// Mitsubishi GX Works2 project: PLCֹ_GROUP_20   PLC: FX3G

// global labels: Global1
VAR_GLOBAL
  Start_Day AT X010 : BOOL;
  Work_Day_Lamp AT Y010 : BOOL;
  Flour_Input AT D1100 : REAL;
  Yeast_Input AT D1110 : REAL;
  Water_Input AT D1120 : REAL;
  Oil_input AT D1130 : REAL;
  Spice_Input AT D1140 : REAL;
  Flour_Container AT D1150 : REAL;
  Yeast_Container AT D1160 : REAL;
  Water_Container AT D1170 : REAL;
  Oil_Container AT D1180 : REAL;
  Spice_Container AT D1190 : REAL;
  Flour_Constant AT E100 : REAL;
  Empty_Flour AT M1 : BOOL;
  Yeast_Ratio AT E0.2 : REAL;
  Water_Ratio AT E0.5 : REAL;
  Oil_Ratio AT E0.3 : REAL;
  Spice_Ratio AT E0.1 : REAL;
  Yeast_Flour_Ratio AT D1200 : REAL;
  Water_Flour_Ratio AT D1210 : REAL;
  Oil_Flour_Ratio AT D1220 : REAL;
  Spice_Flour_Ratio AT D1230 : REAL;
  Out_Of_Stock AT M3 : BOOL;
  Emergency_Stop AT X007 : BOOL;
  End_Of_Day AT M5 : BOOL;
  Const_3secs AT K30 : WORD;
  TC_1 AT TC1 : BOOL;
  TC_3 AT TC3 : BOOL;
  TC_5 AT TC5 : BOOL;
  TS_1 AT TS1 : BOOL;
  TS_5 AT TS5 : BOOL;
  TS_3 AT TS3 : BOOL;
  const_hazi AT K5 : INT;
  TS_9 AT TS9 : BOOL;
  TS_10 AT TS10 : BOOL;
  TS_11 AT TS11 : BOOL;
  TC_9 AT TC9 : BOOL;
  TC_11 AT TC11 : BOOL;
  TC_10 AT TC10 : BOOL;
  Flicker_3secs AT M100 : BOOL;
  Start_Loading_Process AT X002 : BOOL;
  Timer_3s AT TC3 : BOOL;
  Timer_3s_const AT K30 : INT;
  Preparing_Light AT Y005 : BOOL;
  Const_30_Oil AT E30.0 : REAL;
  Const_10_Spice AT E10.0 : REAL;
  Const_100_Flour AT E100.0 : REAL;
  Const_20_Yeast AT E20.0 : REAL;
  Const_50_Water AT E50.0 : REAL;
  Oil_Scale AT D3500 : REAL;
  Spice_Scale AT D3600 : REAL;
  Flour_Scale AT D3200 : REAL;
  Yeast_Scale AT D3300 : REAL;
  Water_Scale AT D3400 : REAL;
  Timer_3s_TS3 AT TS3 : BOOL;
  Kneading_Lamp AT Y001 : BOOL;
  Start_Kneading AT X001 : BOOL;
  Const_210 AT E210.0 : REAL;
  D_Kneading AT D3700 : REAL;
  Start_Proofing AT X011 : BOOL;
  Click_Counter AT CC1 : BOOL;
  Clicks AT K2 : INT;
  Clicks2 AT CS1 : BOOL;
  TC_4 AT TC4 : BOOL;
  Timer_3sec AT K30 : INT;
  Finish_Timer AT TS4 : BOOL;
  Start_Blink AT M300 : BOOL;
  Timer_Blink3 AT K3 : INT;
  Y2_timer AT TS5 : BOOL;
  Lamp_2 AT Y002 : BOOL;
  Lamp_3 AT Y003 : BOOL;
  TC_6 AT TC6 : BOOL;
  Y3_timer AT TS6 : BOOL;
  Finish_Proofing AT M301 : BOOL;
  D_Proofing AT D6000 : REAL;
  Baking_Timer AT TC20 : BOOL;
  Timer_4Secs AT K40 : INT;
  Baking_Lamp AT Y004 : BOOL;
  Y4_Timer AT TS20 : BOOL;
  D_Oven AT D7000 : REAL;
  Checking_Quality AT X003 : BOOL;
  Analog_Input_2 AT D8281 : INT;
  Save_Analog AT D1700 : REAL;
  Const_400 AT E400.0 : REAL;
  Norm_Input AT D1900 : REAL;
  Const_5 AT E2000.0 : REAL;
  Const_1 AT E400.0 : REAL;
  LT_5 AT M123 : BOOL;
  GT_1 AT M127 : BOOL;
  Quality_Lamp AT Y006 : BOOL;
  Timer_5secs AT TC18 : BOOL;
  Timer_5sec AT TS18 : BOOL;
  Const_555 AT K50 : INT;
  D_Shelf AT D5555 : REAL;
  Process_Done AT M63 : BOOL;
  Check_Counter AT CC5 : BOOL;
  Check_Clickes AT K2 : INT;
  Checks AT K2 : INT;
  False_Quality AT M96 : BOOL;
  Quality_Clicks AT CS5 : BOOL;
  Turn_Off_Y1 AT M275 : BOOL;
  Keep_Y1_Work_Right AT M201 : BOOL;
END_VAR

// task Task_01 (event TRUE, interval 0, priority 31): POU_01

PROGRAM POU_01
(* structured ladder/FBD written out as ST: instructions are called as NAME(EN, inputs, outputs); _pN, _eN, _tN stand for wires *)
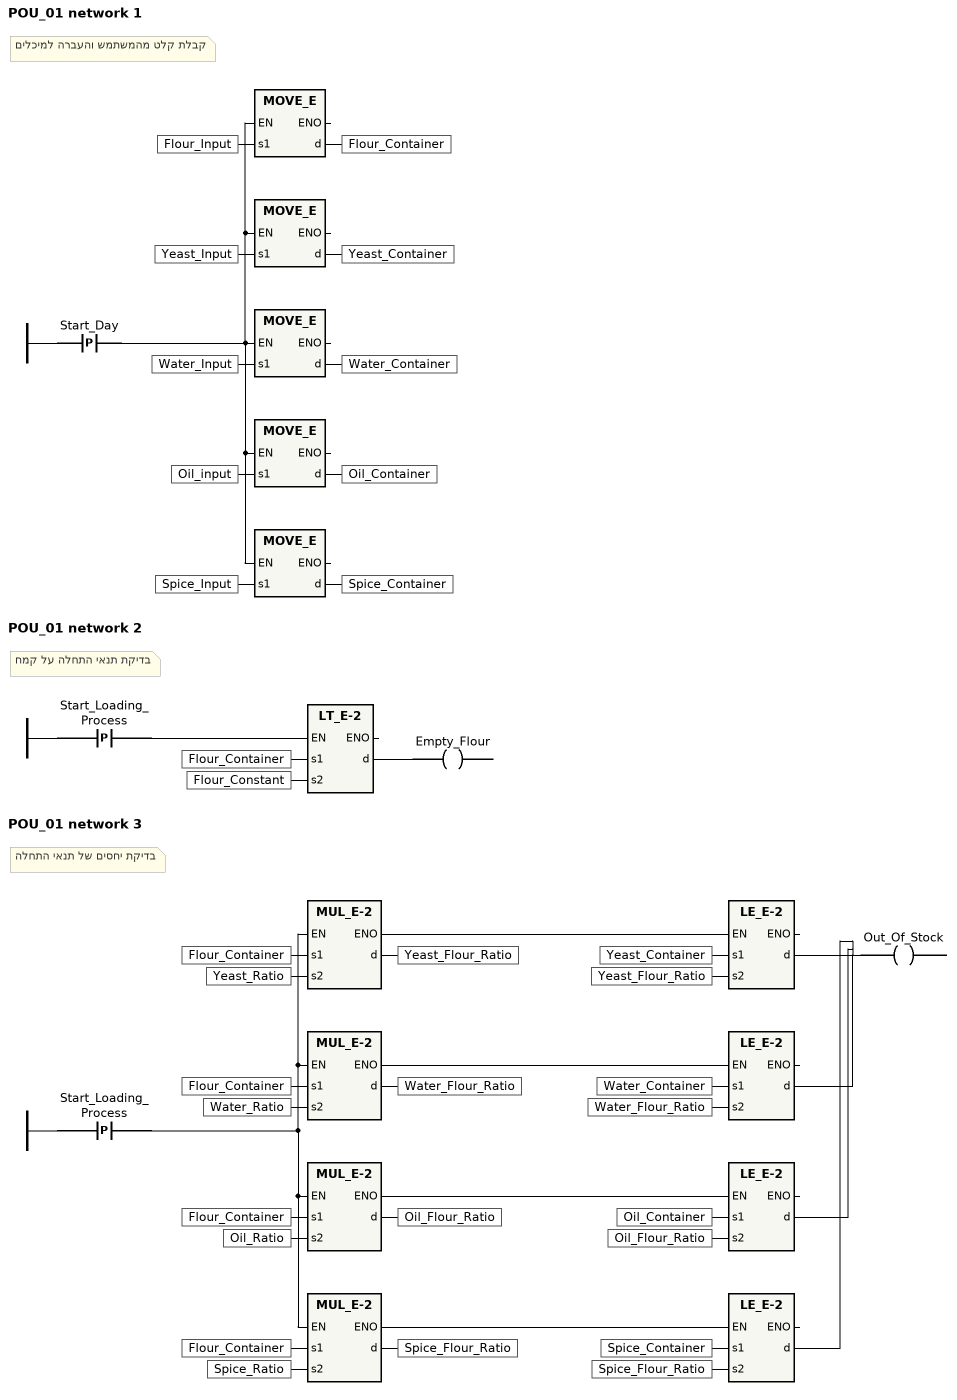
(* network 1 *)
(* קבלת קלט מהמשתמש והעברה למיכלים *)
_p1 := LDP(TRUE, Start_Day);
MOVE_E(_p1, Flour_Input, Flour_Container);
MOVE_E(_p1, Yeast_Input, Yeast_Container);
MOVE_E(_p1, Water_Input, Water_Container);
MOVE_E(_p1, Oil_input, Oil_Container);
MOVE_E(_p1, Spice_Input, Spice_Container);
(* network 2 *)
(* בדיקת תנאי התחלה על קמח *)
LT_E(LDP(TRUE, Start_Loading_Process), Flour_Container, Flour_Constant, _t1);
Empty_Flour := _t1;
(* network 3 *)
(* בדיקת יחסים של תנאי התחלה *)
_p1 := LDP(TRUE, Start_Loading_Process);
_e2 := MUL_E(_p1, Flour_Container, Yeast_Ratio, Yeast_Flour_Ratio);
LE_E(_e2, Yeast_Container, Yeast_Flour_Ratio, _t3);
_e4 := MUL_E(_p1, Flour_Container, Water_Ratio, Water_Flour_Ratio);
LE_E(_e4, Water_Container, Water_Flour_Ratio, _t5);
_e6 := MUL_E(_p1, Flour_Container, Oil_Ratio, Oil_Flour_Ratio);
LE_E(_e6, Oil_Container, Oil_Flour_Ratio, _t7);
_e8 := MUL_E(_p1, Flour_Container, Spice_Ratio, Spice_Flour_Ratio);
LE_E(_e8, Spice_Container, Spice_Flour_Ratio, _t9);
Out_Of_Stock := _t3 OR _t5 OR _t7 OR _t9;
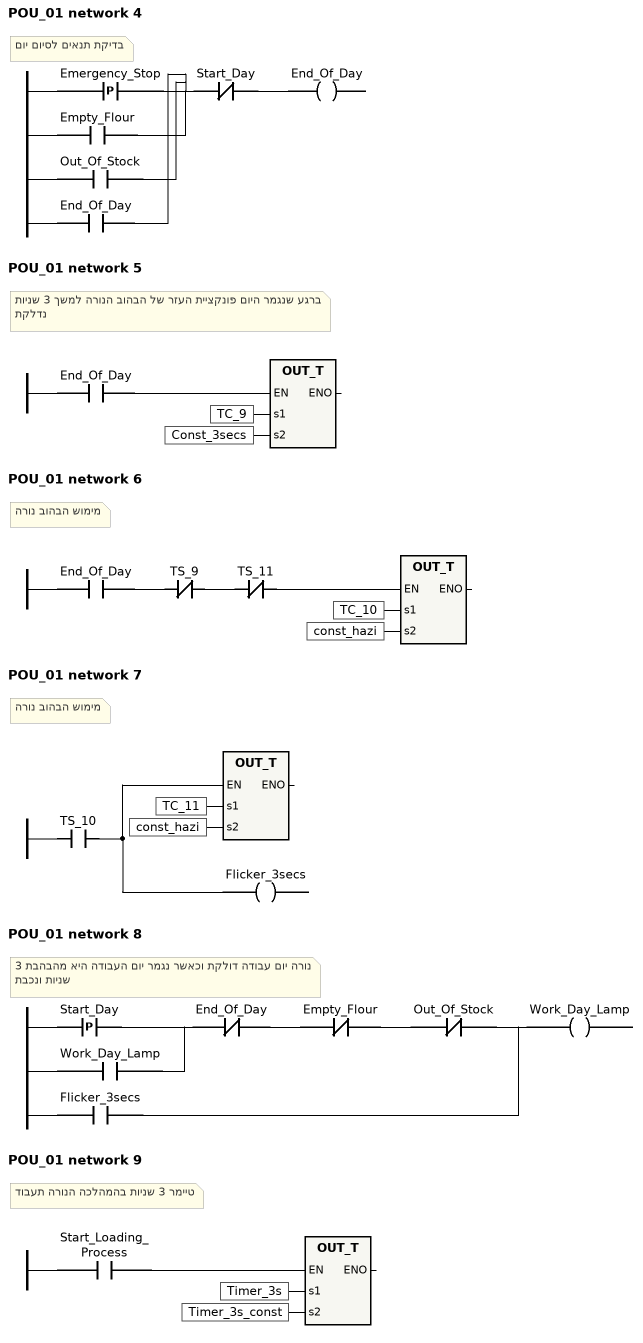
(* network 4 *)
(* בדיקת תנאים לסיום יום *)
End_Of_Day := (LDP(TRUE, Emergency_Stop) OR Empty_Flour OR Out_Of_Stock OR End_Of_Day) AND NOT Start_Day;
(* network 5 *)
(* ברגע שנגמר היום פונקציית העזר של הבהוב הנורה למשך 3 שניות נדלקת *)
OUT_T(End_Of_Day, TC_9, Const_3secs);
(* network 6 *)
(* מימוש הבהוב נורה *)
OUT_T(End_Of_Day AND NOT TS_9 AND NOT TS_11, TC_10, const_hazi);
(* network 7 *)
(* מימוש הבהוב נורה *)
OUT_T(TS_10, TC_11, const_hazi);
Flicker_3secs := TS_10;
(* network 8 *)
(* נורה יום עבודה דולקת וכאשר נגמר יום העבודה היא מהבהבת 3 שניות ונכבת *)
Work_Day_Lamp := ((((LDP(TRUE, Start_Day) OR Work_Day_Lamp) AND NOT End_Of_Day) AND NOT Empty_Flour) AND NOT Out_Of_Stock) OR Flicker_3secs;
(* network 9 *)
(* טיימר 3 שניות בהמהלכה הנורה תעבוד *)
OUT_T(Start_Loading_Process, Timer_3s, Timer_3s_const);
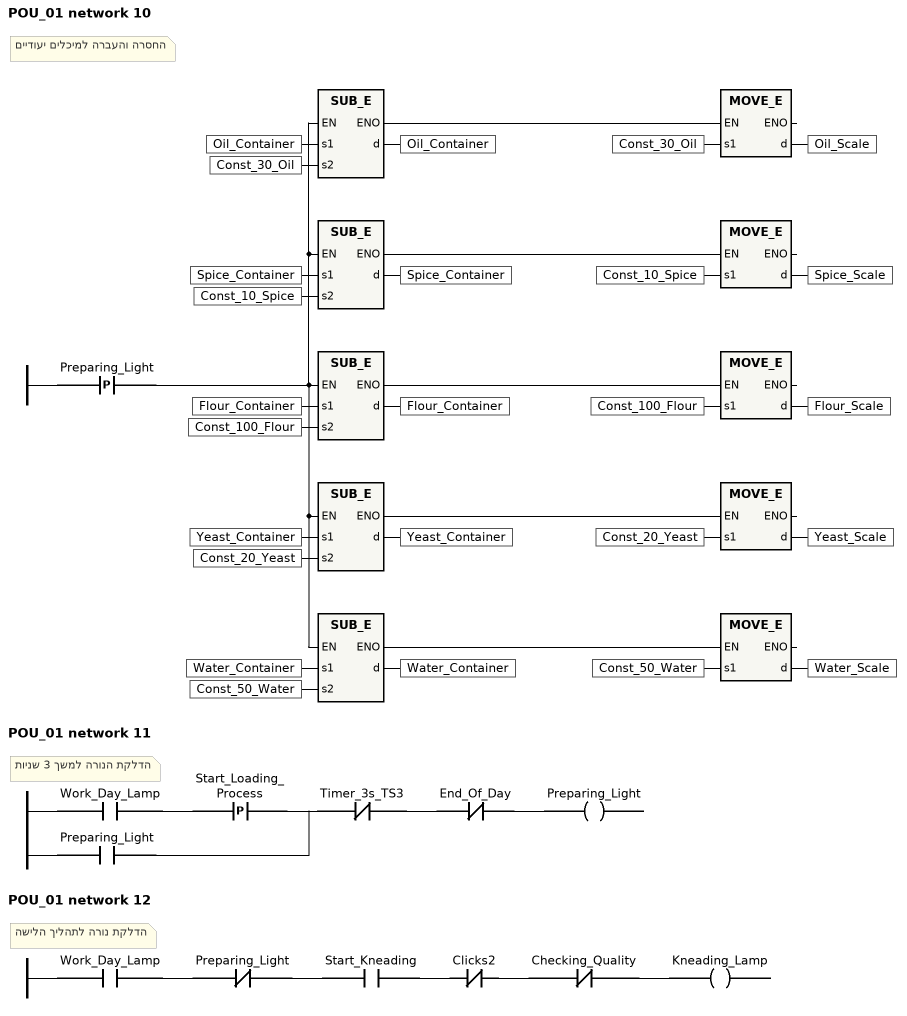
(* network 10 *)
(* החסרה והעברה למיכלים יעודיים *)
_p1 := LDP(TRUE, Preparing_Light);
_e2 := SUB_E(_p1, Oil_Container, Const_30_Oil, Oil_Container);
MOVE_E(_e2, Const_30_Oil, Oil_Scale);
_e3 := SUB_E(_p1, Spice_Container, Const_10_Spice, Spice_Container);
MOVE_E(_e3, Const_10_Spice, Spice_Scale);
_e4 := SUB_E(_p1, Flour_Container, Const_100_Flour, Flour_Container);
MOVE_E(_e4, Const_100_Flour, Flour_Scale);
_e5 := SUB_E(_p1, Yeast_Container, Const_20_Yeast, Yeast_Container);
MOVE_E(_e5, Const_20_Yeast, Yeast_Scale);
_e6 := SUB_E(_p1, Water_Container, Const_50_Water, Water_Container);
MOVE_E(_e6, Const_50_Water, Water_Scale);
(* network 11 *)
(* הדלקת הנורה למשך 3 שניות *)
Preparing_Light := (((Work_Day_Lamp AND LDP(TRUE, Start_Loading_Process)) OR Preparing_Light) AND NOT Timer_3s_TS3) AND NOT End_Of_Day;
(* network 12 *)
(* הדלקת נורה לתהליך הלישה *)
Kneading_Lamp := Work_Day_Lamp AND NOT Preparing_Light AND Start_Kneading AND NOT Clicks2 AND NOT Checking_Quality;
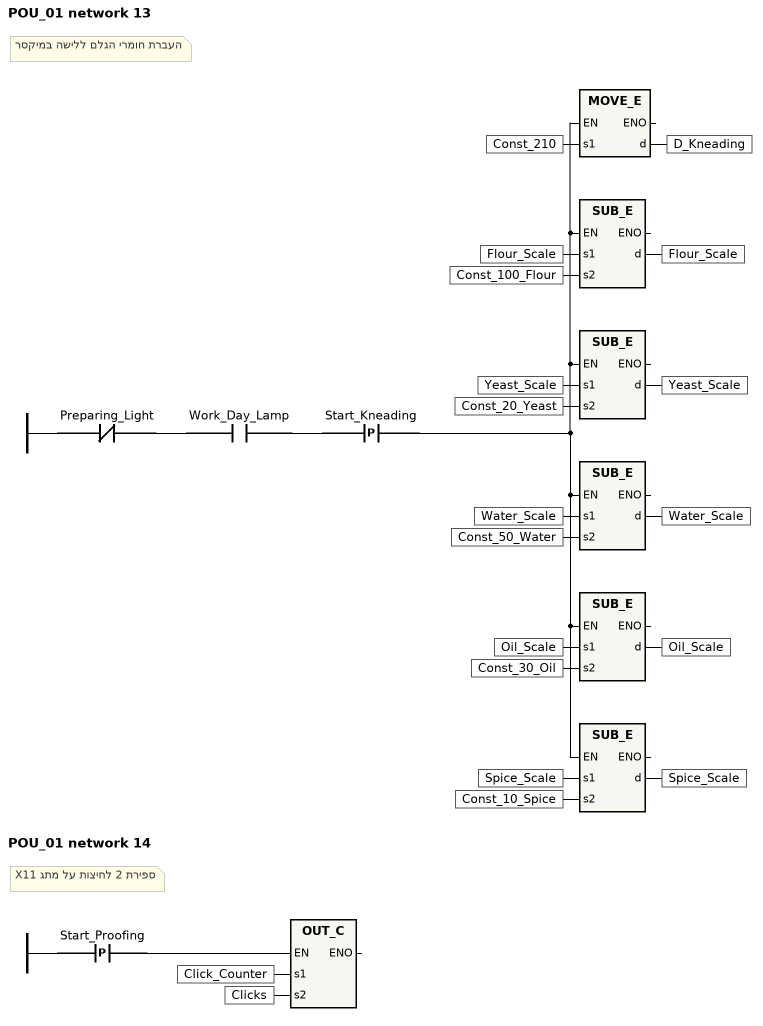
(* network 13 *)
(* העברת חומרי הגלם ללישה במיקסר *)
_p1 := NOT Preparing_Light AND Work_Day_Lamp AND LDP(TRUE, Start_Kneading);
MOVE_E(_p1, Const_210, D_Kneading);
SUB_E(_p1, Flour_Scale, Const_100_Flour, Flour_Scale);
SUB_E(_p1, Yeast_Scale, Const_20_Yeast, Yeast_Scale);
SUB_E(_p1, Water_Scale, Const_50_Water, Water_Scale);
SUB_E(_p1, Oil_Scale, Const_30_Oil, Oil_Scale);
SUB_E(_p1, Spice_Scale, Const_10_Spice, Spice_Scale);
(* network 14 *)
(* ספירת 2 לחיצות על מתג X11 *)
OUT_C(LDP(TRUE, Start_Proofing), Click_Counter, Clicks);
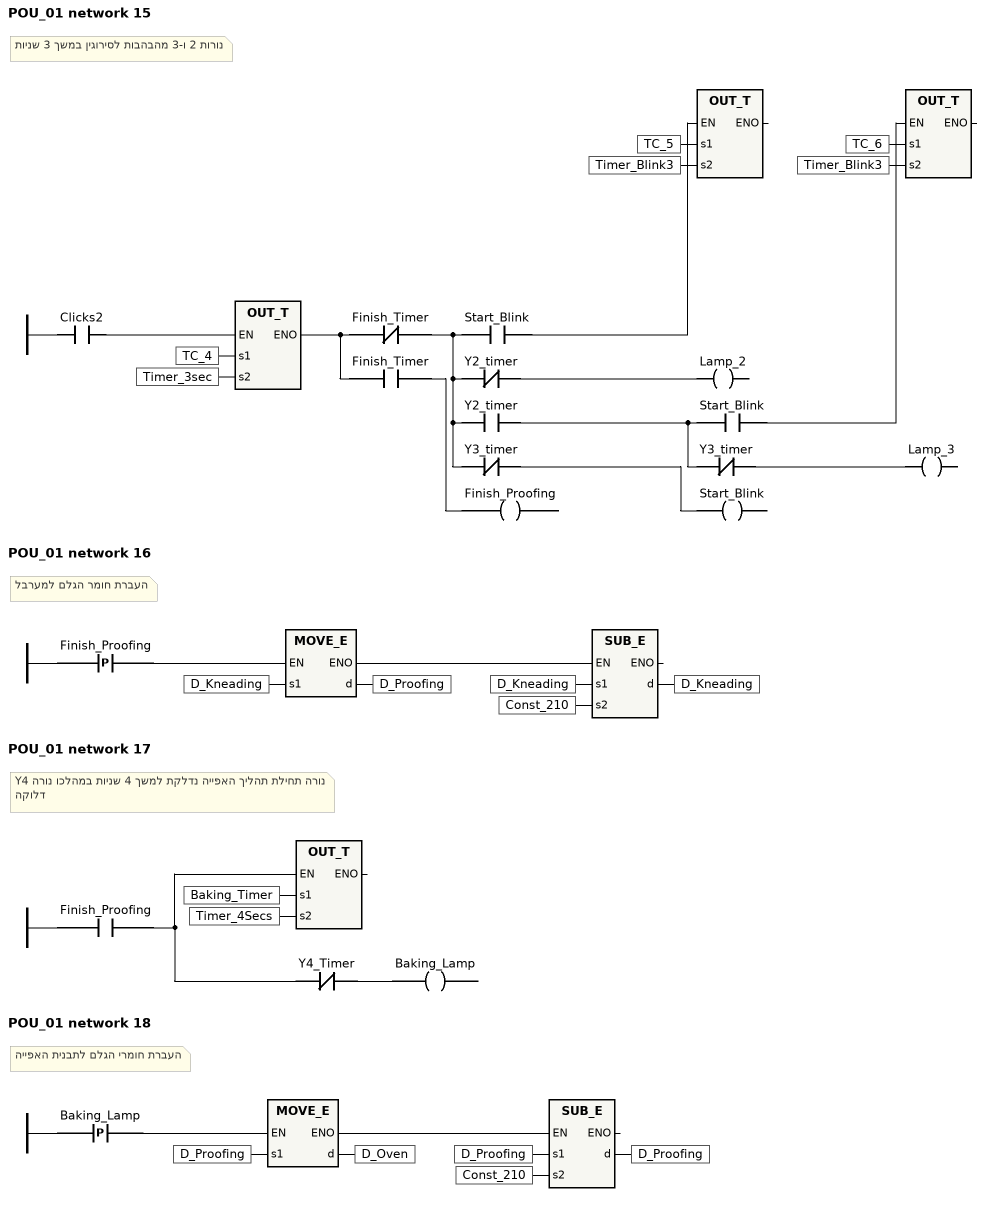
(* network 15 *)
(* נורות 2 ו-3 מהבהבות לסירוגין במשך 3 שניות *)
_e1 := OUT_T(Clicks2, TC_4, Timer_3sec);
_p2 := _e1 AND NOT Finish_Timer;
OUT_T(_p2 AND Start_Blink, TC_5, Timer_Blink3);
Lamp_2 := _p2 AND NOT Y2_timer;
_p3 := _p2 AND Y2_timer;
OUT_T(_p3 AND Start_Blink, TC_6, Timer_Blink3);
Lamp_3 := _p3 AND NOT Y3_timer;
Start_Blink := _p2 AND NOT Y3_timer;
Finish_Proofing := _e1 AND Finish_Timer;
(* network 16 *)
(* העברת חומר הגלם למערבל *)
_e1 := MOVE_E(LDP(TRUE, Finish_Proofing), D_Kneading, D_Proofing);
SUB_E(_e1, D_Kneading, Const_210, D_Kneading);
(* network 17 *)
(* נורה תחילת תהליך האפייה נדלקת למשך 4 שניות במהלכו נורה Y4 דלוקה *)
OUT_T(Finish_Proofing, Baking_Timer, Timer_4Secs);
Baking_Lamp := Finish_Proofing AND NOT Y4_Timer;
(* network 18 *)
(* העברת חומרי הגלם לתבנית האפייה *)
_e1 := MOVE_E(LDP(TRUE, Baking_Lamp), D_Proofing, D_Oven);
SUB_E(_e1, D_Proofing, Const_210, D_Proofing);
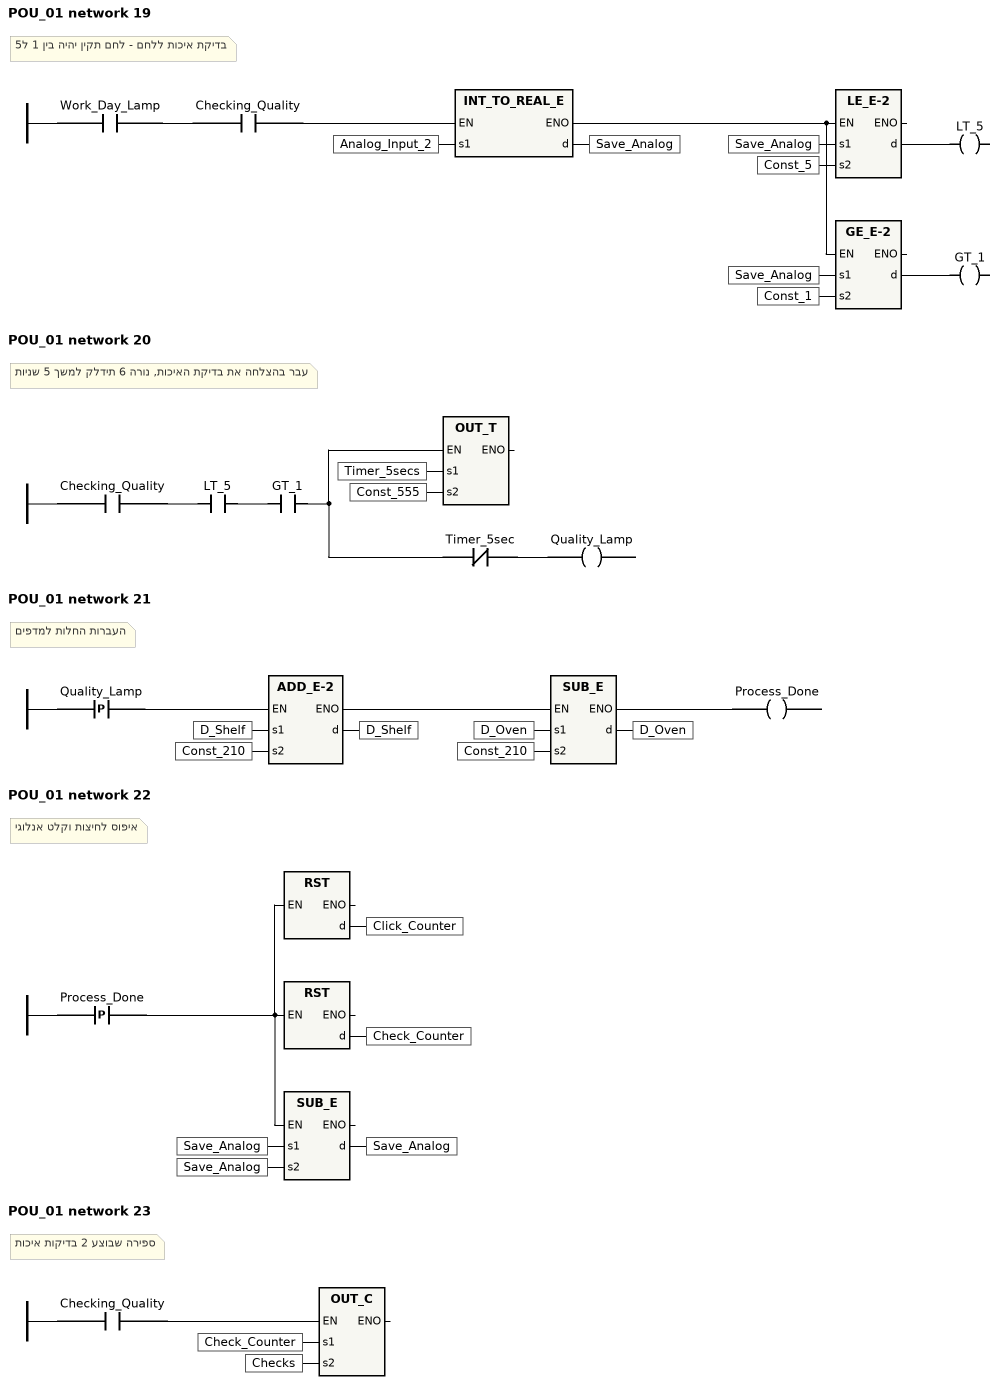
(* network 19 *)
(* בדיקת איכות ללחם - לחם תקין יהיה בין 1 ל5 *)
_e1 := INT_TO_REAL_E(Work_Day_Lamp AND Checking_Quality, Analog_Input_2, Save_Analog);
LE_E(_e1, Save_Analog, Const_5, _t2);
LT_5 := _t2;
GE_E(_e1, Save_Analog, Const_1, _t3);
GT_1 := _t3;
(* network 20 *)
(* עבר בהצלחה את בדיקת האיכות, נורה 6 תידלק למשך 5 שניות *)
_p1 := Checking_Quality AND LT_5 AND GT_1;
OUT_T(_p1, Timer_5secs, Const_555);
Quality_Lamp := _p1 AND NOT Timer_5sec;
(* network 21 *)
(* העברות החלות למדפים *)
_e1 := ADD_E(LDP(TRUE, Quality_Lamp), D_Shelf, Const_210, D_Shelf);
_e2 := SUB_E(_e1, D_Oven, Const_210, D_Oven);
Process_Done := _e2;
(* network 22 *)
(* איפוס לחיצות וקלט אנלוגי *)
_p1 := LDP(TRUE, Process_Done);
RST(_p1, Click_Counter);
RST(_p1, Check_Counter);
SUB_E(_p1, Save_Analog, Save_Analog, Save_Analog);
(* network 23 *)
(* ספירה שבוצע 2 בדיקות איכות *)
OUT_C(Checking_Quality, Check_Counter, Checks);
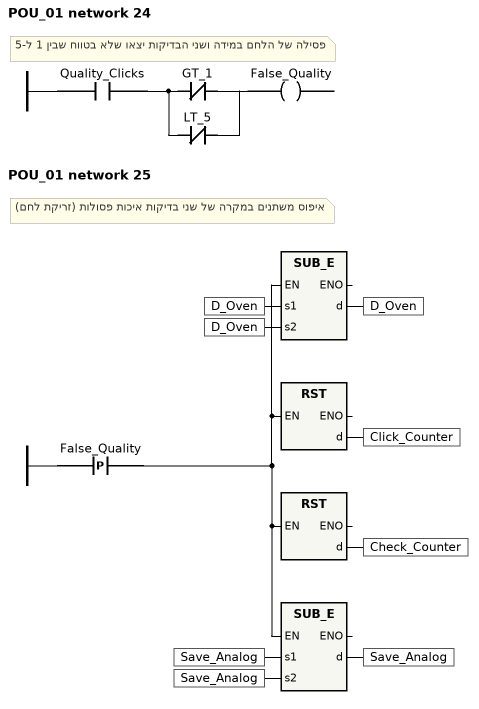
(* network 24 *)
(* פסילה של הלחם במידה ושני הבדיקות יצאו שלא בטווח שבין 1 ל-5 *)
False_Quality := (Quality_Clicks AND NOT GT_1) OR (Quality_Clicks AND NOT LT_5);
(* network 25 *)
(* איפוס משתנים במקרה של שני בדיקות איכות פסולות (זריקת לחם) *)
_p1 := LDP(TRUE, False_Quality);
SUB_E(_p1, D_Oven, D_Oven, D_Oven);
RST(_p1, Click_Counter);
RST(_p1, Check_Counter);
SUB_E(_p1, Save_Analog, Save_Analog, Save_Analog);
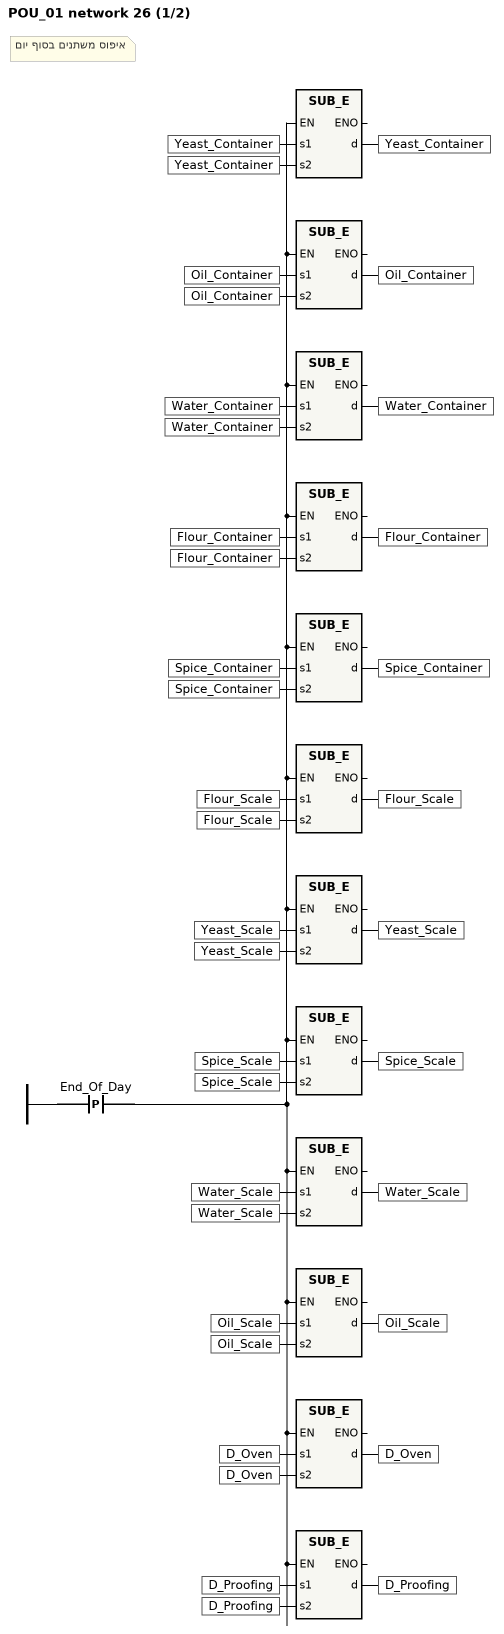
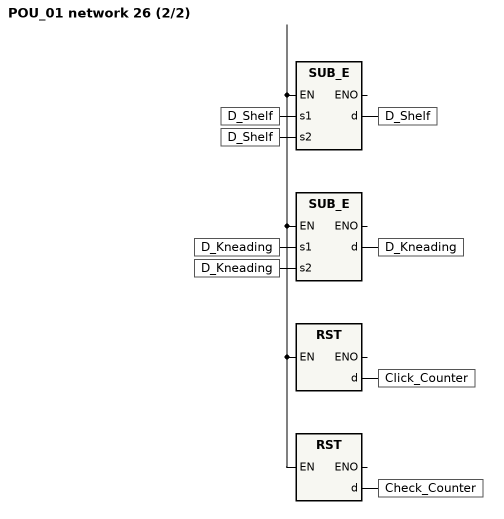
(* network 26 *)
(* איפוס משתנים בסוף יום *)
_p1 := LDP(TRUE, End_Of_Day);
SUB_E(_p1, Yeast_Container, Yeast_Container, Yeast_Container);
SUB_E(_p1, Oil_Container, Oil_Container, Oil_Container);
SUB_E(_p1, Water_Container, Water_Container, Water_Container);
SUB_E(_p1, Flour_Container, Flour_Container, Flour_Container);
SUB_E(_p1, Spice_Container, Spice_Container, Spice_Container);
SUB_E(_p1, Flour_Scale, Flour_Scale, Flour_Scale);
SUB_E(_p1, Yeast_Scale, Yeast_Scale, Yeast_Scale);
SUB_E(_p1, Spice_Scale, Spice_Scale, Spice_Scale);
SUB_E(_p1, Water_Scale, Water_Scale, Water_Scale);
SUB_E(_p1, Oil_Scale, Oil_Scale, Oil_Scale);
SUB_E(_p1, D_Oven, D_Oven, D_Oven);
SUB_E(_p1, D_Proofing, D_Proofing, D_Proofing);
SUB_E(_p1, D_Shelf, D_Shelf, D_Shelf);
SUB_E(_p1, D_Kneading, D_Kneading, D_Kneading);
RST(_p1, Click_Counter);
RST(_p1, Check_Counter);
END_PROGRAM
